SYSTEM System (* System Configuration *)
  (* Standard: 61499-1 *)
  (* Version 0.0, 7/8/2016, Andrei, nxtControl GmbH *)
  APPLICATION APP1
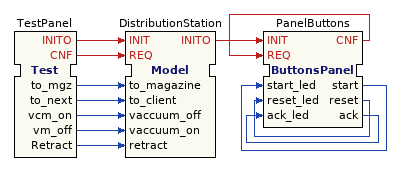
    FBS
      DistributionStation : Model;
      TestPanel : Test;
      PanelButtons : ButtonsPanel;
    END_FBS
    EVENT_CONNECTIONS
      TestPanel.INITO TO DistributionStation.INIT;
      TestPanel.CNF TO DistributionStation.REQ;
      DistributionStation.INITO TO PanelButtons.INIT;
      PanelButtons.CNF TO PanelButtons.REQ;
    END_CONNECTIONS
    DATA_CONNECTIONS
      TestPanel.to_mgz TO DistributionStation.to_magazine;
      TestPanel.to_next TO DistributionStation.to_client;
      TestPanel.vcm_on TO DistributionStation.vaccuum_off;
      TestPanel.vm_off TO DistributionStation.vaccuum_on;
      TestPanel.Retract TO DistributionStation.retract;
      PanelButtons.start TO PanelButtons.start_led;
      PanelButtons.reset TO PanelButtons.reset_led;
      PanelButtons.ack TO PanelButtons.ack_led;
    END_CONNECTIONS
  END_APPLICATION
  APPLICATION DistributingStation
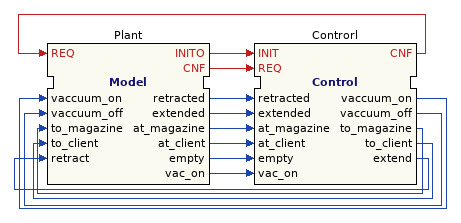
    FBS
      Plant : Model;
      Controrl : Control;
    END_FBS
    EVENT_CONNECTIONS
      Plant.INITO TO Controrl.INIT;
      Plant.CNF TO Controrl.REQ;
      Controrl.CNF TO Plant.REQ;
    END_CONNECTIONS
    DATA_CONNECTIONS
      Plant.retracted TO Controrl.retracted;
      Plant.extended TO Controrl.extended;
      Plant.at_magazine TO Controrl.at_magazine;
      Plant.at_client TO Controrl.at_client;
      Plant.empty TO Controrl.empty;
      Controrl.vaccuum_on TO Plant.vaccuum_on;
      Controrl.vaccuum_off TO Plant.vaccuum_off;
      Controrl.to_magazine TO Plant.to_magazine;
      Controrl.to_client TO Plant.to_client;
      Controrl.extend TO Plant.retract;
      Plant.vac_on TO Controrl.vac_on;
    END_CONNECTIONS
  END_APPLICATION
  APPLICATION RefactoredDS
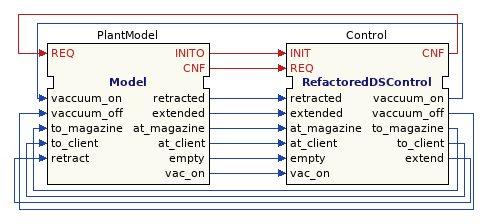
    FBS
      PlantModel : Model;
      Control : RefactoredDSControl;
    END_FBS
    EVENT_CONNECTIONS
      PlantModel.INITO TO Control.INIT;
      PlantModel.CNF TO Control.REQ;
      Control.CNF TO PlantModel.REQ;
    END_CONNECTIONS
    DATA_CONNECTIONS
      PlantModel.retracted TO Control.retracted;
      PlantModel.extended TO Control.extended;
      PlantModel.at_magazine TO Control.at_magazine;
      PlantModel.at_client TO Control.at_client;
      PlantModel.empty TO Control.empty;
      PlantModel.vac_on TO Control.vac_on;
      Control.vaccuum_on TO PlantModel.vaccuum_on;
      Control.vaccuum_off TO PlantModel.vaccuum_off;
      Control.to_magazine TO PlantModel.to_magazine;
      Control.to_client TO PlantModel.to_client;
      Control.extend TO PlantModel.retract;
    END_CONNECTIONS
  END_APPLICATION
  DEVICE DSHMI : NXT_RMTDEV
    RESOURCE RES0 : EMB_RES_ENH(PRIO := 0)
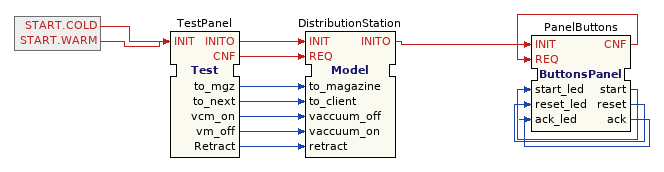
      FBS
        DistributionStation : Model;
        TestPanel : Test;
        PanelButtons : ButtonsPanel;
      END_FBS
      EVENT_CONNECTIONS
        TestPanel.INITO TO DistributionStation.INIT;
        TestPanel.CNF TO DistributionStation.REQ;
        START.COLD TO TestPanel.INIT;
        START.WARM TO TestPanel.INIT;
        DistributionStation.INITO TO PanelButtons.INIT;
        PanelButtons.CNF TO PanelButtons.REQ;
      END_CONNECTIONS
      DATA_CONNECTIONS
        TestPanel.to_mgz TO DistributionStation.to_magazine;
        TestPanel.to_next TO DistributionStation.to_client;
        TestPanel.vcm_on TO DistributionStation.vaccuum_off;
        TestPanel.vm_off TO DistributionStation.vaccuum_on;
        TestPanel.Retract TO DistributionStation.retract;
        PanelButtons.start TO PanelButtons.start_led;
        PanelButtons.reset TO PanelButtons.reset_led;
        PanelButtons.ack TO PanelButtons.ack_led;
      END_CONNECTIONS
    END_RESOURCE
  END_DEVICE
  DEVICE DS : NXT_RMTDEV(MGR_ID := "127.0.0.1:61499", HMI_ID := "127.0.0.1:61498", WATCH_ID := "127.0.0.1:61497")
    RESOURCE RES0 : EMB_RES_ENH
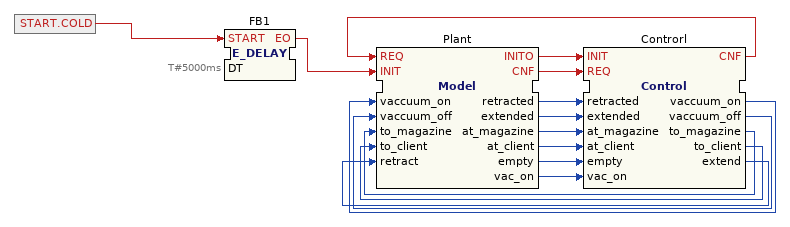
      FBS
        Plant : Model;
        Controrl : Control;
        FB1 : E_DELAY(DT := T#5000ms);
      END_FBS
      EVENT_CONNECTIONS
        Plant.INITO TO Controrl.INIT;
        Plant.CNF TO Controrl.REQ;
        Controrl.CNF TO Plant.REQ;
        START.COLD TO FB1.START;
        FB1.EO TO Plant.INIT;
      END_CONNECTIONS
      DATA_CONNECTIONS
        Plant.retracted TO Controrl.retracted;
        Plant.extended TO Controrl.extended;
        Plant.at_magazine TO Controrl.at_magazine;
        Plant.at_client TO Controrl.at_client;
        Plant.empty TO Controrl.empty;
        Controrl.vaccuum_on TO Plant.vaccuum_on;
        Controrl.vaccuum_off TO Plant.vaccuum_off;
        Controrl.to_magazine TO Plant.to_magazine;
        Controrl.to_client TO Plant.to_client;
        Controrl.extend TO Plant.retract;
        Plant.vac_on TO Controrl.vac_on;
      END_CONNECTIONS
    END_RESOURCE
  END_DEVICE
  DEVICE RDS : NXT_RMTDEV(MGR_ID := "127.0.0.1:61499", HMI_ID := "127.0.0.1:61498", WATCH_ID := "127.0.0.1:61497")
    RESOURCE RES0 : EMB_RES_ENH
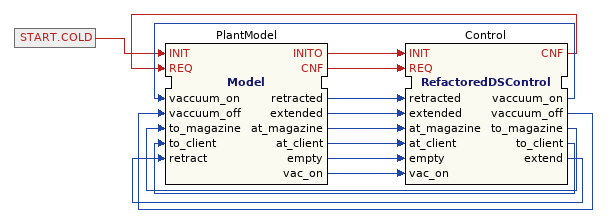
      FBS
        PlantModel : Model;
        Control : RefactoredDSControl;
      END_FBS
      EVENT_CONNECTIONS
        PlantModel.INITO TO Control.INIT;
        PlantModel.CNF TO Control.REQ;
        START.COLD TO PlantModel.INIT;
        Control.CNF TO PlantModel.REQ;
      END_CONNECTIONS
      DATA_CONNECTIONS
        PlantModel.retracted TO Control.retracted;
        PlantModel.extended TO Control.extended;
        PlantModel.at_magazine TO Control.at_magazine;
        PlantModel.at_client TO Control.at_client;
        PlantModel.empty TO Control.empty;
        PlantModel.vac_on TO Control.vac_on;
        Control.vaccuum_on TO PlantModel.vaccuum_on;
        Control.vaccuum_off TO PlantModel.vaccuum_off;
        Control.to_magazine TO PlantModel.to_magazine;
        Control.to_client TO PlantModel.to_client;
        Control.extend TO PlantModel.retract;
      END_CONNECTIONS
    END_RESOURCE
  END_DEVICE
  MAPPINGS
    APP1.DistributionStation ON DSHMI.RES0;
    APP1.TestPanel ON DSHMI.RES0;
    APP1.PanelButtons ON DSHMI.RES0;
    DistributingStation.Plant ON DS.RES0;
    DistributingStation.Controrl ON DS.RES0;
    RefactoredDS.PlantModel ON RDS.RES0;
    RefactoredDS.Control ON RDS.RES0;
  END_MAPPINGS
END_SYSTEM
